PROGRAM P_DALI2_Test
VAR
	fbStarCount: FB_DALI253QueryControlGearStartCounter(0);
	bStart: BOOL;
	nAddress: BYTE := 10;
	eAddressType: Tc3_DALI.E_DALIAddressType := Tc3_DALI.E_DALIAddressType.Short;
	eCommandPriority: Tc3_DALI.E_DALICommandPriority := Tc3_DALI.E_DALICommandPriority.Middle;
	nControlGearStartCounter: UDINT;
END_VAR

VAR CONSTANT
	DALI_LINE_NUM: INT := 1;
END_VAR

fbStarCount.ipDALICommunication := P_DALI_Background.arrfbKL6821Communication[DALI_LINE_NUM];


fbStarCount(
	bError=> , 
	ipResultMessage=> , 
	bStart:= bStart, 
	nAddress:= nAddress, 
	eAddressType:= eAddressType, 
	eCommandPriority:=eCommandPriority , 
	bBusy=> , 
	nControlGearStartCounter=> nControlGearStartCounter);

END_PROGRAM

(* stored: Version 1.1.0.1
   POU P_DALI2_Test: Id {3db5867d-1fd4-40c6-a0d5-1e3c9d8d57cb}, SpecialFunc None *)
